// TwinCAT 3 PLC project RT1
// ProgramVersion: 3.1.4024.0
// libraries:
//   Tc2_Standard, * (Beckhoff Automation GmbH)
//   Tc2_System, * (Beckhoff Automation GmbH)
//   Tc3_Module, * (Beckhoff Automation GmbH)
// project tree:
//   / GlobalTextList.TcGTLO, PlcTask.TcTTO, Visualization Manager.TcVMO (not stored), VISU_TASK.TcTTO
//   POUs/ MAIN.TcPOU
//   SimulationComps/ FB_CylinderSimul.TcPOU
//   VISUs/ CylSimul.TcVIS, Visualization.TcVIS
// real-time tasks:
//   TASK PlcTask: cycle T#10ms, priority 20, ADS port 350
//   TASK PlcTask1: cycle T#10ms, priority 21, ADS port 351
//   TASK VISU_TASK: cycle T#200000us, priority 30, ADS port 352
// I/O:
//   DEVICE Device 1 (EtherCAT) (disabled), AmsNetId 169.254.34.75.2.1
//     Term 1 (EK1100) [EK1100 EtherCAT Coupler (2A E-Bus)]
//       Term 2 (EL1008) [EL1008 8Ch. Dig. Input 24V, 3ms]
//       Term 3 (EL2004) [EL2004 4Ch. Dig. Output 24V, 0.5A]

CONFIGURATION RT1
    RESOURCE PLC ON TwinCAT3
        TASK PlcTask(INTERVAL := T#10ms, PRIORITY := 20);
        TASK VISU_TASK(INTERVAL := T#200000us, PRIORITY := 30);
        PROGRAM MAIN WITH PlcTask : MAIN;
        PROGRAM VisuElems_Visu_Prg WITH VISU_TASK : VisuElems.Visu_Prg;
    END_RESOURCE
END_CONFIGURATION

// ---- POUs/MAIN.TcPOU
PROGRAM MAIN
VAR
	offSet AT %Q*:LREAL;
	cilindro:FB_CylinderSimul;
	avanca AT %I*: BOOL;
	recua AT %I*: BOOL;
	sensorFwd	AT %Q*: BOOL;
	sensorBwd	at %Q*: BOOL;
END_VAR

cilindro(
	moveFwd:=avanca , 
	moveBwd:= recua, 
	course:= 500, 
	moveVel:= 100, 
	cycleTime:= T#10MS, 
	sensorCylFwd=> sensorFwd, 
	sensorCylBwd=> sensorBwd, 
	currentPos=> , 
	posPercent=> offSet);

END_PROGRAM

// ---- SimulationComps/FB_CylinderSimul.TcPOU
FUNCTION_BLOCK FB_CylinderSimul
VAR_INPUT
	moveFwd: BOOL;
	moveBwd: BOOL;
	course:LREAL:=500;	//cylinder course in mm
	moveVel:LREAL:=100;	//move velocity in mm/s
	cycleTime:TIME:=T#10MS;
END_VAR
VAR_OUTPUT
	sensorCylFwd: BOOL;
	sensorCylBwd: BOOL;
	currentPos:LREAL;
	posPercent:LREAL;
END_VAR
VAR
	movementPerCycle: LREAL;
END_VAR

movementPerCycle:= TIME_TO_LREAL(cycletime)/1000*moveVel;
IF moveFwd AND NOT moveBwd THEN
	m_CylFwd();
ELSIF moveBwd AND NOT moveFwd THEN
	m_CylBwd();
END_IF

sensorCylBwd:= currentPos <= 1;
sensorCylFwd:= currentPos >= (course - 1);

METHOD m_CylBwd : BOOL
VAR_INPUT
END_VAR
currentPos:= LIMIT(0,currentPos-movementPerCycle,course);
posPercent:= currentPos*100/course;
END_METHOD

METHOD m_CylFwd : BOOL
VAR_INPUT
END_VAR
currentPos:= LIMIT(0,currentPos+movementPerCycle,course);
posPercent:= currentPos*100/course;
END_METHOD

END_FUNCTION_BLOCK

// ---- VISUs/CylSimul.TcVIS
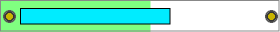
VISUALIZATION CylSimul  // 280x32
VAR_IN_OUT
	currPosPercent:LREAL;
	sensorFwd: BOOL;
	sensorBwd: BOOL;
END_VAR
    Rectangle (0,0 150x32)
    Rectangle (20,8 150x16)
        p3528305787: currPosPercent
        p874137650: currPosPercent
    Lamp1 (2,9 15x15), variable: sensorBwd, style: Lamp-Lamp1-Yellow
    Lamp1 (264,9 15x15), variable: sensorFwd, style: Lamp-Lamp1-Yellow
END_VISUALIZATION

// ---- VISUs/Visualization.TcVIS
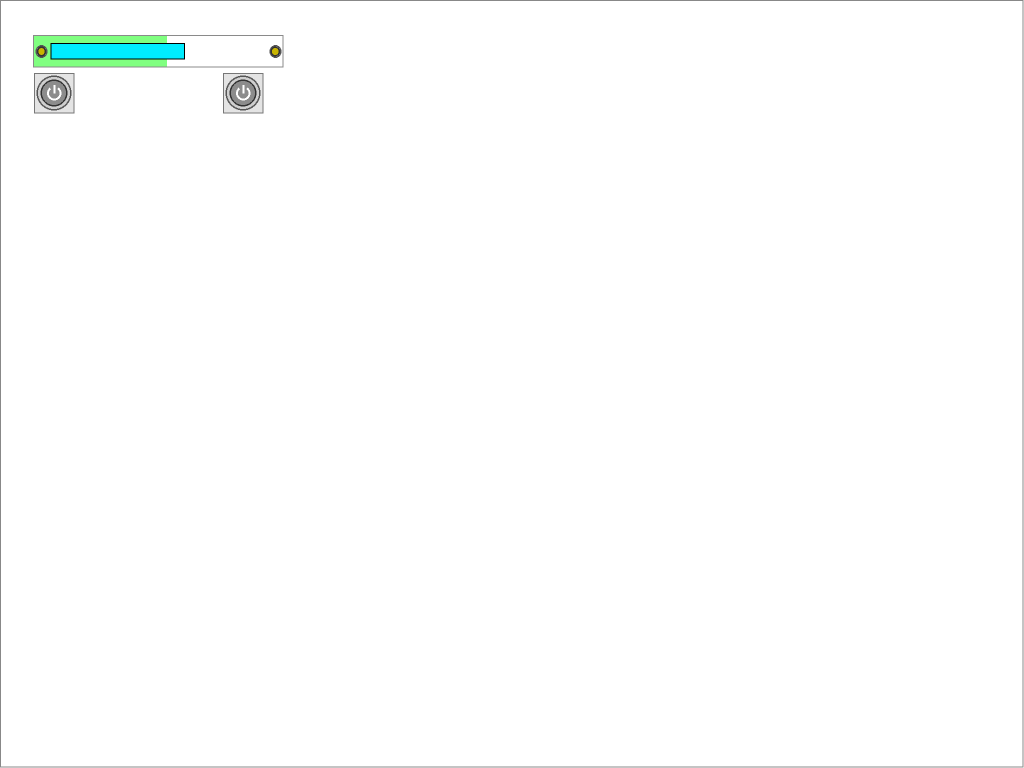
VISUALIZATION Visualization  // 1024x768
    Frame (33,35 250x32)
        shows CylSimul(currPosPercent := MAIN.offSet, sensorFwd := MAIN.sensorFwd, sensorBwd := MAIN.sensorBwd)
    PowerSwitch (34,73 40x40), variable: MAIN.recua, behaviour: TAP, style: Switch-PowerSwitch-Gray
    PowerSwitch (223,73 40x40), variable: MAIN.avanca, behaviour: TAP, style: Switch-PowerSwitch-Gray
END_VISUALIZATION
